TYPE EtcMasterBase_62654B43 :
STRUCT
END_STRUCT
END_TYPE
